FUNCTION_BLOCK FB_CondensingBoiler EXTENDS FB_Actuator2Point
VAR_INPUT
END_VAR
VAR_OUTPUT
END_VAR
VAR
	//I/O Links
	bSetStatusOn_OUT 	AT %Q* : BOOL := FALSE;
END_VAR

SelectControlMode();

//input states may be read via LON connector - not implemented yet

METHOD SetState_BO : BOOL
VAR_INPUT
END_VAR
//output
bSetStatusOn_OUT := bSetStatusOn;
END_METHOD

END_FUNCTION_BLOCK

(* stored: Version 1.1.0.1, ProductVersion 3.1.4024.10
   POU FB_CondensingBoiler: Id {532a516d-9cc8-4820-b59b-bc9ad3e263f3}, SpecialFunc None
   Method SetState_BO: Id {fa4c4620-aa78-459b-9cb0-16279b461c9a} *)
